// TIA Portal V17 export
// export: Created 2025-06-20T10:18:27.4190976Z, ExportSetting WithDefaults, DisplayName Totally Integrated Automation Portal, DisplayVersion V17 Update 8, DisplayName TIA Portal Openness, DisplayVersion V17 Update 8, DisplayName TIA Portal Version Control Interface, DisplayVersion V17, DisplayName SINAMICS Startdrive Advanced, DisplayVersion V17 SP2, DisplayName SINAMICS Startdrive G110M, G120, G120C, G120D, G120P, G115D, DisplayVersion V17 SP2, DisplayName SINAMICS Startdrive G130, G150, S120, S150, SINAMICS MV, S210, DisplayVersion V17 SP2, DisplayName STEP 7 Professional, DisplayVersion V17 Update 8, DisplayName SINUMERIK ONE STEP 7 Toolbox, DisplayVersion V17 Update 12, DisplayName SINUMERIK ONE PLC Basic Program Plus, DisplayVersion V17 Update 12, DisplayName SINUMERIK 840D sl STEP 7 Toolbox, DisplayVersion V17 Update 12, DisplayName STEP 7 Safety, DisplayVersion V17 Update 6, DisplayName WinCC Advanced, DisplayVersion V17 Update 8
DATA_BLOCK "DB17000_MAINTENANCE_GLOBAL_VARIABLES"   // DB17000
{ S7_Optimized_Access := 'TRUE'; DB_Accessible_From_OPC_UA := 'FALSE' }
VERSION : 0.1
// stored: AutoNumber false, DBAccessibleFromOPCUA false, DBAccessibleFromWebserver true, IsOnlyStoredInLoadMemory false, IsRetainMemResEnabled false, IsWriteProtectedInAS false, MemoryReserve 100
   VAR
      ACTION_DONE : Struct
         POWDER : Struct
            UNIT_1 : Struct
               GENERAL : Struct
                  POWDER_TUBE_SECTION_4 : Bool;
                  POWDER_TUBE_SECTION_5 : Bool;
                  RIGID_TUBE_OF_SPLITTER : Bool;
                  COMBINER_MEDICOAT_CALIBRATION : Bool;
                  NOZZLE_MEDICOAT_CALIBRATION : Bool;
                  POWDER_FLOW_OBTAINING : Bool;
               END_STRUCT;
               HOPPER_1 : Struct
                  HOPPER : Bool;
                  MEDICOAT_CALIBRATION : Bool;
                  PINCH_VALVE : Bool;
                  TUBE_SECTION_1 : Bool;
                  TUBE_SECTION_2 : Bool;
                  LOAD_CELLS : Bool;
               END_STRUCT;
               HOPPER_2 : Struct
                  HOPPER : Bool;
                  MEDICOAT_CALIBRATION : Bool;
                  PINCH_VALVE : Bool;
                  TUBE_SECTION_1 : Bool;
                  TUBE_SECTION_2 : Bool;
                  LOAD_CELLS : Bool;
               END_STRUCT;
               FEEDER_1 : Struct
                  COMPLET_FEEDER_REPLACEMENT : Bool;
                  HOPPER_L1 : Bool;
                  TUBE_SECTION_3_L1 : Bool;
                  HOPPER_L2 : Bool;
                  TUBE_SECTION_3_L2 : Bool;
                  TIGHTNESS_TEST_L1 : Bool;
                  TIGHTNESS_TEST_L2 : Bool;
                  MEDICOAT_L1 : Bool;
                  MEDICOAT_L2 : Bool;
               END_STRUCT;
            END_STRUCT;
            UNIT_2 : Struct
               GENERAL : Struct
                  POWDER_TUBE_SECTION_4 : Bool;
                  POWDER_TUBE_SECTION_5 : Bool;
                  RIGID_TUBE_OF_SPLITTER : Bool;
                  COMBINER_MEDICOAT_CALIBRATION : Bool;
                  NOZZLE_MEDICOAT_CALIBRATION : Bool;
                  POWDER_FLOW_OBTAINING : Bool;
               END_STRUCT;
               HOPPER_1 : Struct
                  HOPPER : Bool;
                  MEDICOAT_CALIBRATION : Bool;
                  PINCH_VALVE : Bool;
                  TUBE_SECTION_1 : Bool;
                  TUBE_SECTION_2 : Bool;
                  LOAD_CELLS : Bool;
               END_STRUCT;
               HOPPER_2 : Struct
                  HOPPER : Bool;
                  MEDICOAT_CALIBRATION : Bool;
                  PINCH_VALVE : Bool;
                  TUBE_SECTION_1 : Bool;
                  TUBE_SECTION_2 : Bool;
                  LOAD_CELLS : Bool;
               END_STRUCT;
               HOPPER_3 : Struct
                  HOPPER : Bool;
                  MEDICOAT_CALIBRATION : Bool;
                  PINCH_VALVE : Bool;
                  TUBE_SECTION_1 : Bool;
                  TUBE_SECTION_2 : Bool;
                  LOAD_CELLS : Bool;
               END_STRUCT;
               FEEDER_1 : Struct
                  COMPLET_FEEDER_REPLACEMENT : Bool;
                  HOPPER_L1 : Bool;
                  TUBE_SECTION_3_L1 : Bool;
                  HOPPER_L2 : Bool;
                  TUBE_SECTION_3_L2 : Bool;
                  TIGHTNESS_TEST_L1 : Bool;
                  TIGHTNESS_TEST_L2 : Bool;
                  MEDICOAT_L1 : Bool;
                  MEDICOAT_L2 : Bool;
               END_STRUCT;
               FEEDER_2 : Struct
                  COMPLET_FEEDER_REPLACEMENT : Bool;
                  HOPPER_L2 : Bool;
                  TUBE_SECTION_3_L2 : Bool;
                  TIGHTNESS_TEST_L2 : Bool;
                  MEDICOAT_L2 : Bool;
               END_STRUCT;
            END_STRUCT;
         END_STRUCT;
         MACHINE : Struct
            UNIT_1 : Struct
               GENERAL : Struct
                  FIXTURE_1_MODIFICATION : Bool;
                  FIXTURE_2_MODIFICATION : Bool;
                  FIXTURE_3_MODIFICATION : Bool;
                  FIXTURE_4_MODIFICATION : Bool;
                  SEALING_SYSTEM_ST3 : Bool;
                  LASER_HEAD_ADJUSTMENT : Bool;
                  CAMERA : Bool;
                  PROFILOMETER_CALIBRATING : Bool;
                  PROFILOMETER_LENS_CLEANING : Bool;
                  PYROMETER_CONFIG_IN_PROGRESS : Bool;
                  WATER_SYSTEM : Bool;
                  GAS_SYSTEM : Bool;
                  AXIS_REFERENCE_SEQUENCE : Bool;
                  ADJUSTMENT_AXIS_C11 : Bool;
                  ADJUSTMENT_AXIS_C12 : Bool;
                  ADJUSTMENT_AXIS_C13 : Bool;
                  ADJUSTMENT_AXIS_C14 : Bool;
                  ADJUSTMENT_AXIS_X13 : Bool;
                  ADJUSTMENT_AXIS_Z13 : Bool;
                  ADJUSTMENT_AXIS_E10 : Bool;
               END_STRUCT;
               LASER : Struct
                  PROCESS_PROTECTION_GLASS : Bool;
                  FIBRE_PROTECTION_GLASS : Bool;
                  NOZZLE : Bool;
               END_STRUCT;
            END_STRUCT;
            UNIT_2 : Struct
               GENERAL : Struct
                  FIXTURE_1_MODIFICATION : Bool;
                  FIXTURE_2_MODIFICATION : Bool;
                  FIXTURE_3_MODIFICATION : Bool;
                  FIXTURE_4_MODIFICATION : Bool;
                  SEALING_SYSTEM_ST3 : Bool;
                  LASER_HEAD_ADJUSTMENT : Bool;
                  CAMERA : Bool;
                  PROFILOMETER_CALIBRATING : Bool;
                  PROFILOMETER_LENS_CLEANING : Bool;
                  PYROMETER_CONFIG_IN_PROGRESS : Bool;
                  WATER_SYSTEM : Bool;
                  GAS_SYSTEM : Bool;
                  AXIS_REFERENCE_SEQUENCE : Bool;
                  ADJUSTMENT_AXIS_C21 : Bool;
                  ADJUSTMENT_AXIS_C22 : Bool;
                  ADJUSTMENT_AXIS_C23 : Bool;
                  ADJUSTMENT_AXIS_C24 : Bool;
                  ADJUSTMENT_AXIS_X23 : Bool;
                  ADJUSTMENT_AXIS_Z23 : Bool;
                  ADJUSTMENT_AXIS_E20 : Bool;
               END_STRUCT;
               LASER : Struct
                  PROCESS_PROTECTION_GLASS : Bool;
                  FIBRE_PROTECTION_GLASS : Bool;
                  NOZZLE : Bool;
               END_STRUCT;
            END_STRUCT;
         END_STRUCT;
         CELL : Struct
            LOAD_CELL_PART_ROTATION_1 : Bool;
            LOAD_CELL_PART_ROTATION_2 : Bool;
            LOAD_CELL_PART_ROTATION_3 : Bool;
         END_STRUCT;
      END_STRUCT;
      START_REQ_TIMER : TON_TIME;   // START REQUEST TIMER
   END_VAR
BEGIN
   START_REQ_TIMER.PT := T#2S;
END_DATA_BLOCK
